TYPE "pnioSubnetStatus"
TITLE = Type:"PNIO subnet status"
VERSION : 0.1
//["version","date","author","description"],
//["v1.0","2022-10-12","cyanezf","First version"]
   STRUCT
      state : Int;   // Current state
      error : Int;   // Current error
      device { S7_SetPoint := 'False'} : Array[0..1023] of "pnioDeviceStatus";   // Devices
   END_STRUCT;

END_TYPE

